// TIA Portal V16 export
// export: Created 2023-05-15T10:42:05.211121Z, ExportSetting WithDefaults, DisplayName Totally Integrated Automation Portal, DisplayVersion V16 Update 3, DisplayName TIA Portal Version Control Interface, DisplayVersion V16 Update 2, DisplayName TIA Portal Openness, DisplayVersion V16 Update 3, DisplayName SINAMICS Startdrive Advanced, DisplayVersion V16, DisplayName SINAMICS Startdrive G130, G150, S120, S150, SINAMICS MV, S210, DisplayVersion V16, DisplayName SINAMICS Startdrive G110M, G120, G120C, G120D, G120P, DisplayVersion V16, DisplayName STEP 7 Professional, DisplayVersion V16 Update 3, DisplayName STEP 7 Safety, DisplayVersion V16, DisplayName WinCC Advanced, DisplayVersion V16 Update 3
FUNCTION "AUTO_HBA2" : Void   // FC45, LAD
{ S7_Optimized_Access := 'FALSE' }
VERSION : 0.1
// prueba con paco de comit 2 b
// 1040 desde paco
// stored: AutoNumber false, IsIECCheckEnabled false, SetENOAutomatically false, UDAEnableTagReadback false
   VAR_TEMP
      SEGUIR : Bool;
      aux_int_1 : Int;
      TEMP0 : Bool;
   END_VAR
   VAR_TEMP   // added for the SCL form of the ladder/FBD networks
      _w1 : Bool;
      _s5time1 : S5Time;
   END_VAR
BEGIN

REGION Network 1: ACTIVACION VAN300
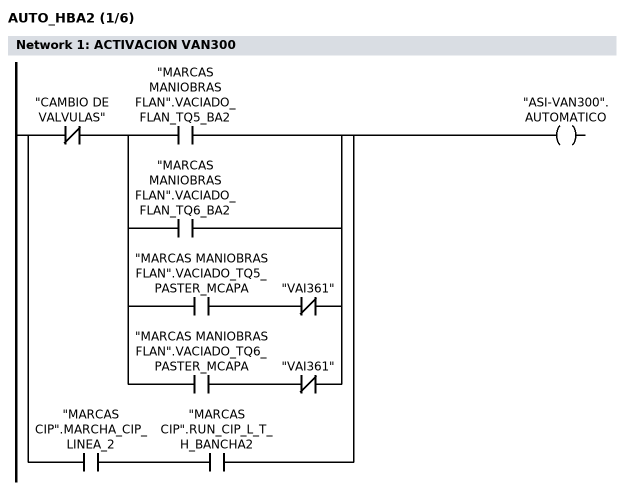
   RUNG wire#powerrail
      I_Contact( "CAMBIO DE VALVULAS" )
      wire#w1
      Contact( "MARCAS MANIOBRAS FLAN".VACIADO_FLAN_TQ5_BA2 )
      wire#w2
      Coil( "ASI-VAN300".AUTOMATICO )
   END_RUNG
   RUNG wire#w1
      Contact( "MARCAS MANIOBRAS FLAN".VACIADO_FLAN_TQ6_BA2 )
   END_RUNG wire#w2
   RUNG wire#w1
      Contact( "MARCAS MANIOBRAS FLAN".VACIADO_TQ5_PASTER_MCAPA )
      I_Contact( "VAI361" )
   END_RUNG wire#w2
   RUNG wire#w1
      Contact( "MARCAS MANIOBRAS FLAN".VACIADO_TQ6_PASTER_MCAPA )
      I_Contact( "VAI361" )
   END_RUNG wire#w2
   RUNG wire#powerrail
      Contact( "MARCAS CIP".MARCHA_CIP_LINEA_2 )
      Contact( "MARCAS CIP".RUN_CIP_L_T_H_BANCHA2 )
   END_RUNG wire#w2
   // the same network as SCL:
   "ASI-VAN300".AUTOMATICO := (NOT "CAMBIO DE VALVULAS" AND ("MARCAS MANIOBRAS FLAN".VACIADO_FLAN_TQ5_BA2 OR "MARCAS MANIOBRAS FLAN".VACIADO_FLAN_TQ6_BA2 OR ("MARCAS MANIOBRAS FLAN".VACIADO_TQ5_PASTER_MCAPA AND NOT "VAI361") OR ("MARCAS MANIOBRAS FLAN".VACIADO_TQ6_PASTER_MCAPA AND NOT "VAI361"))) OR ("MARCAS CIP".MARCHA_CIP_LINEA_2 AND "MARCAS CIP".RUN_CIP_L_T_H_BANCHA2);
END_REGION

REGION Network 2: ACTIVACION VMN301
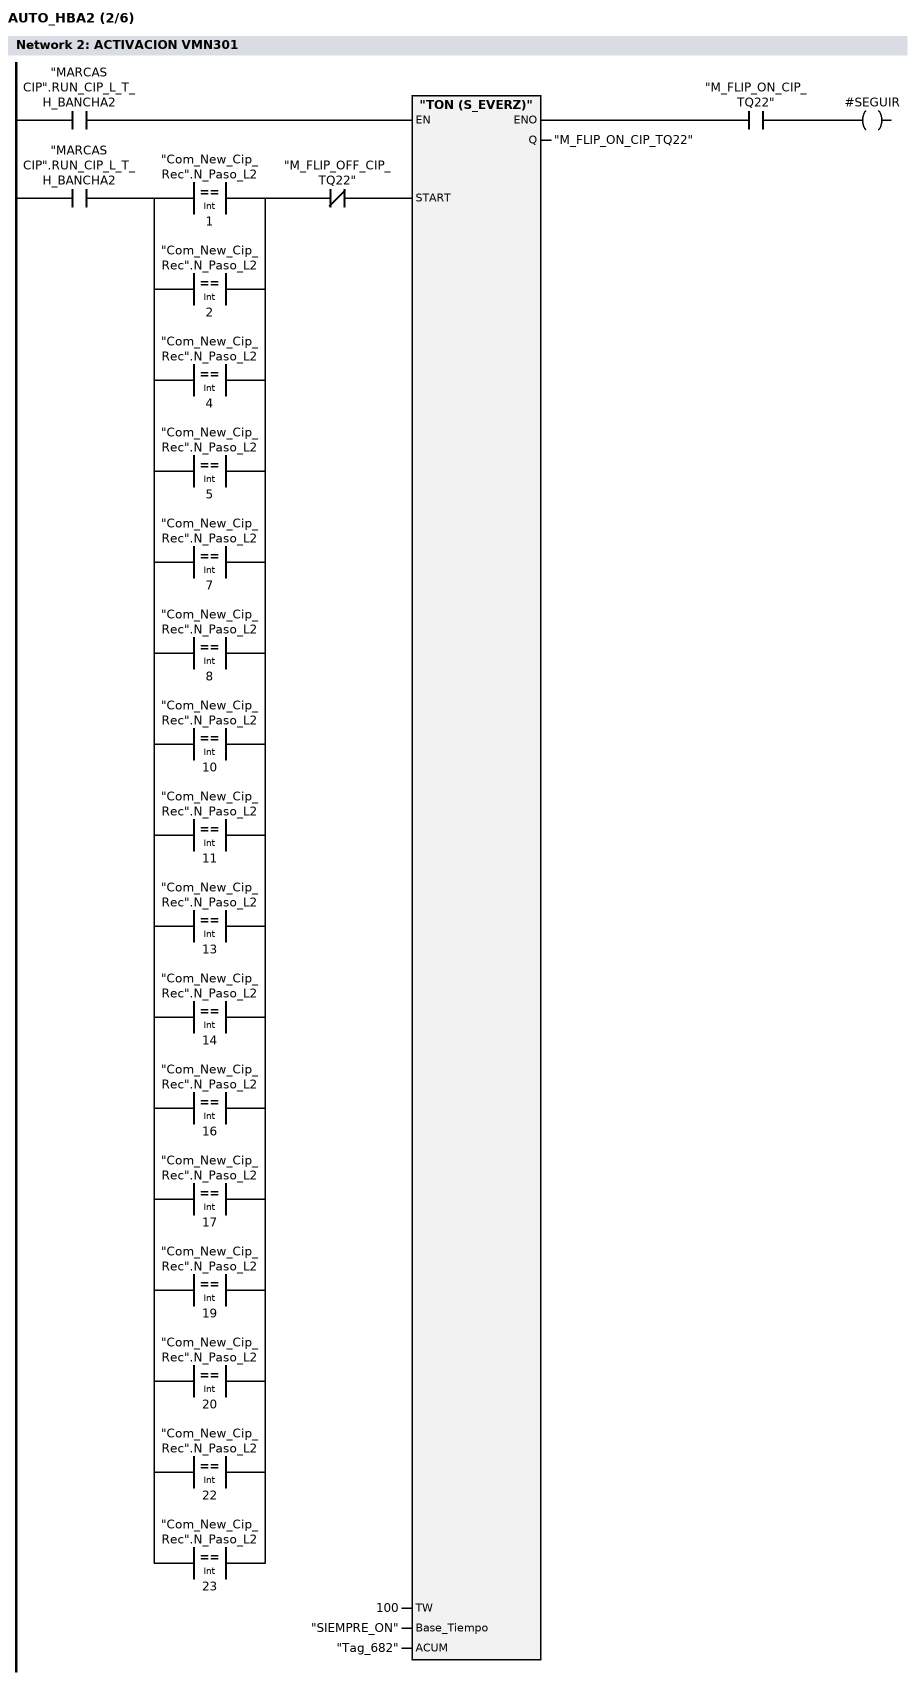
   RUNG wire#powerrail
      Contact( "MARCAS CIP".RUN_CIP_L_T_H_BANCHA2 )
      "TON (S_EVERZ)"(TW := 100, Base_Tiempo := "SIEMPRE_ON", Q => "M_FLIP_ON_CIP_TQ22", ACUM := "Tag_682", START := wire#w3)
      Contact( "M_FLIP_ON_CIP_TQ22" )
      Coil( #SEGUIR )
   END_RUNG
   RUNG wire#powerrail
      Contact( "MARCAS CIP".RUN_CIP_L_T_H_BANCHA2 )
      wire#w1
      { S7_Templates := "SrcType := Int" } EQ_Contact(in1 := "Com_New_Cip_Rec".N_Paso_L2, in2 := 1)
      wire#w2
      I_Contact( "M_FLIP_OFF_CIP_TQ22" )
   END_RUNG wire#w3
   RUNG wire#w1
      { S7_Templates := "SrcType := Int" } EQ_Contact(in1 := "Com_New_Cip_Rec".N_Paso_L2, in2 := 2)
   END_RUNG wire#w2
   RUNG wire#w1
      { S7_Templates := "SrcType := Int" } EQ_Contact(in1 := "Com_New_Cip_Rec".N_Paso_L2, in2 := 4)
   END_RUNG wire#w2
   RUNG wire#w1
      { S7_Templates := "SrcType := Int" } EQ_Contact(in1 := "Com_New_Cip_Rec".N_Paso_L2, in2 := 5)
   END_RUNG wire#w2
   RUNG wire#w1
      { S7_Templates := "SrcType := Int" } EQ_Contact(in1 := "Com_New_Cip_Rec".N_Paso_L2, in2 := 7)
   END_RUNG wire#w2
   RUNG wire#w1
      { S7_Templates := "SrcType := Int" } EQ_Contact(in1 := "Com_New_Cip_Rec".N_Paso_L2, in2 := 8)
   END_RUNG wire#w2
   RUNG wire#w1
      { S7_Templates := "SrcType := Int" } EQ_Contact(in1 := "Com_New_Cip_Rec".N_Paso_L2, in2 := 10)
   END_RUNG wire#w2
   RUNG wire#w1
      { S7_Templates := "SrcType := Int" } EQ_Contact(in1 := "Com_New_Cip_Rec".N_Paso_L2, in2 := 11)
   END_RUNG wire#w2
   RUNG wire#w1
      { S7_Templates := "SrcType := Int" } EQ_Contact(in1 := "Com_New_Cip_Rec".N_Paso_L2, in2 := 13)
   END_RUNG wire#w2
   RUNG wire#w1
      { S7_Templates := "SrcType := Int" } EQ_Contact(in1 := "Com_New_Cip_Rec".N_Paso_L2, in2 := 14)
   END_RUNG wire#w2
   RUNG wire#w1
      { S7_Templates := "SrcType := Int" } EQ_Contact(in1 := "Com_New_Cip_Rec".N_Paso_L2, in2 := 16)
   END_RUNG wire#w2
   RUNG wire#w1
      { S7_Templates := "SrcType := Int" } EQ_Contact(in1 := "Com_New_Cip_Rec".N_Paso_L2, in2 := 17)
   END_RUNG wire#w2
   RUNG wire#w1
      { S7_Templates := "SrcType := Int" } EQ_Contact(in1 := "Com_New_Cip_Rec".N_Paso_L2, in2 := 19)
   END_RUNG wire#w2
   RUNG wire#w1
      { S7_Templates := "SrcType := Int" } EQ_Contact(in1 := "Com_New_Cip_Rec".N_Paso_L2, in2 := 20)
   END_RUNG wire#w2
   RUNG wire#w1
      { S7_Templates := "SrcType := Int" } EQ_Contact(in1 := "Com_New_Cip_Rec".N_Paso_L2, in2 := 22)
   END_RUNG wire#w2
   RUNG wire#w1
      { S7_Templates := "SrcType := Int" } EQ_Contact(in1 := "Com_New_Cip_Rec".N_Paso_L2, in2 := 23)
   END_RUNG wire#w2
   // the same network as SCL:
   "TON (S_EVERZ)"(EN := "MARCAS CIP".RUN_CIP_L_T_H_BANCHA2,
                   START := "MARCAS CIP".RUN_CIP_L_T_H_BANCHA2 AND (("Com_New_Cip_Rec".N_Paso_L2 = 1) OR ("Com_New_Cip_Rec".N_Paso_L2 = 2) OR ("Com_New_Cip_Rec".N_Paso_L2 = 4) OR ("Com_New_Cip_Rec".N_Paso_L2 = 5) OR ("Com_New_Cip_Rec".N_Paso_L2 = 7) OR ("Com_New_Cip_Rec".N_Paso_L2 = 8) OR ("Com_New_Cip_Rec".N_Paso_L2 = 10) OR ("Com_New_Cip_Rec".N_Paso_L2 = 11) OR ("Com_New_Cip_Rec".N_Paso_L2 = 13) OR ("Com_New_Cip_Rec".N_Paso_L2 = 14) OR ("Com_New_Cip_Rec".N_Paso_L2 = 16) OR ("Com_New_Cip_Rec".N_Paso_L2 = 17) OR ("Com_New_Cip_Rec".N_Paso_L2 = 19) OR ("Com_New_Cip_Rec".N_Paso_L2 = 20) OR ("Com_New_Cip_Rec".N_Paso_L2 = 22) OR ("Com_New_Cip_Rec".N_Paso_L2 = 23)) AND NOT "M_FLIP_OFF_CIP_TQ22",
                   TW := 100,
                   Base_Tiempo := "SIEMPRE_ON",
                   ACUM := "Tag_682",
                   Q => "M_FLIP_ON_CIP_TQ22",
                   ENO => #_w1);
   #SEGUIR := #_w1 AND "M_FLIP_ON_CIP_TQ22";
END_REGION

REGION Network 3
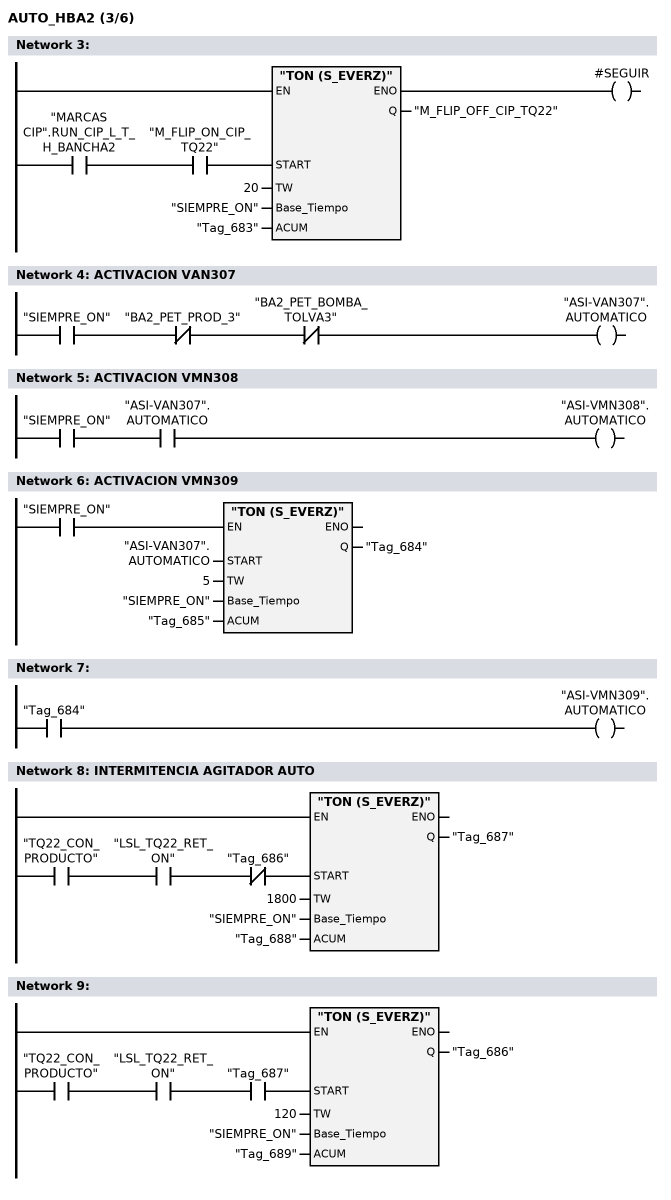
   RUNG wire#powerrail
      "TON (S_EVERZ)"(TW := 20, Base_Tiempo := "SIEMPRE_ON", Q => "M_FLIP_OFF_CIP_TQ22", ACUM := "Tag_683", START := wire#w1)
      Coil( #SEGUIR )
   END_RUNG
   RUNG wire#powerrail
      Contact( "MARCAS CIP".RUN_CIP_L_T_H_BANCHA2 )
      Contact( "M_FLIP_ON_CIP_TQ22" )
   END_RUNG wire#w1
   // the same network as SCL:
   "TON (S_EVERZ)"(START := "MARCAS CIP".RUN_CIP_L_T_H_BANCHA2 AND "M_FLIP_ON_CIP_TQ22",
                   TW := 20,
                   Base_Tiempo := "SIEMPRE_ON",
                   ACUM := "Tag_683",
                   Q => "M_FLIP_OFF_CIP_TQ22",
                   ENO => #_w1);
   #SEGUIR := #_w1;
END_REGION

REGION Network 4: ACTIVACION VAN307
   RUNG wire#powerrail
      Contact( "SIEMPRE_ON" )
      I_Contact( "BA2_PET_PROD_3" )
      I_Contact( "BA2_PET_BOMBA_TOLVA3" )
      Coil( "ASI-VAN307".AUTOMATICO )
   END_RUNG
   // the same network as SCL:
   "ASI-VAN307".AUTOMATICO := "SIEMPRE_ON" AND NOT "BA2_PET_PROD_3" AND NOT "BA2_PET_BOMBA_TOLVA3";
END_REGION

REGION Network 5: ACTIVACION VMN308
   RUNG wire#powerrail
      Contact( "SIEMPRE_ON" )
      Contact( "ASI-VAN307".AUTOMATICO )
      Coil( "ASI-VMN308".AUTOMATICO )
   END_RUNG
   // the same network as SCL:
   "ASI-VMN308".AUTOMATICO := "SIEMPRE_ON" AND "ASI-VAN307".AUTOMATICO;
END_REGION

REGION Network 6: ACTIVACION VMN309
   RUNG wire#powerrail
      Contact( "SIEMPRE_ON" )
      "TON (S_EVERZ)"(START := "ASI-VAN307".AUTOMATICO, TW := 5, Base_Tiempo := "SIEMPRE_ON", Q => "Tag_684", ACUM := "Tag_685")
   END_RUNG
   // the same network as SCL:
   IF "SIEMPRE_ON" THEN
       "TON (S_EVERZ)"(START := "ASI-VAN307".AUTOMATICO,
                       TW := 5,
                       Base_Tiempo := "SIEMPRE_ON",
                       ACUM := "Tag_685",
                       Q => "Tag_684");
   END_IF;
END_REGION

REGION Network 7
   RUNG wire#powerrail
      Contact( "Tag_684" )
      Coil( "ASI-VMN309".AUTOMATICO )
   END_RUNG
   // the same network as SCL:
   "ASI-VMN309".AUTOMATICO := "Tag_684";
END_REGION

REGION Network 8: INTERMITENCIA AGITADOR AUTO
   RUNG wire#powerrail
      "TON (S_EVERZ)"(TW := 1800, Base_Tiempo := "SIEMPRE_ON", Q => "Tag_687", ACUM := "Tag_688", START := wire#w1)
   END_RUNG
   RUNG wire#powerrail
      Contact( "TQ22_CON_PRODUCTO" )
      Contact( "LSL_TQ22_RET_ON" )
      I_Contact( "Tag_686" )
   END_RUNG wire#w1
   // the same network as SCL:
   "TON (S_EVERZ)"(START := "TQ22_CON_PRODUCTO" AND "LSL_TQ22_RET_ON" AND NOT "Tag_686",
                   TW := 1800,
                   Base_Tiempo := "SIEMPRE_ON",
                   ACUM := "Tag_688",
                   Q => "Tag_687");
END_REGION

REGION Network 9
   RUNG wire#powerrail
      "TON (S_EVERZ)"(TW := 120, Base_Tiempo := "SIEMPRE_ON", Q => "Tag_686", ACUM := "Tag_689", START := wire#w1)
   END_RUNG
   RUNG wire#powerrail
      Contact( "TQ22_CON_PRODUCTO" )
      Contact( "LSL_TQ22_RET_ON" )
      Contact( "Tag_687" )
   END_RUNG wire#w1
   // the same network as SCL:
   "TON (S_EVERZ)"(START := "TQ22_CON_PRODUCTO" AND "LSL_TQ22_RET_ON" AND "Tag_687",
                   TW := 120,
                   Base_Tiempo := "SIEMPRE_ON",
                   ACUM := "Tag_689",
                   Q => "Tag_686");
END_REGION

REGION Network 10: ACTIVACION AGITADOR TQ22 (NUEVO)
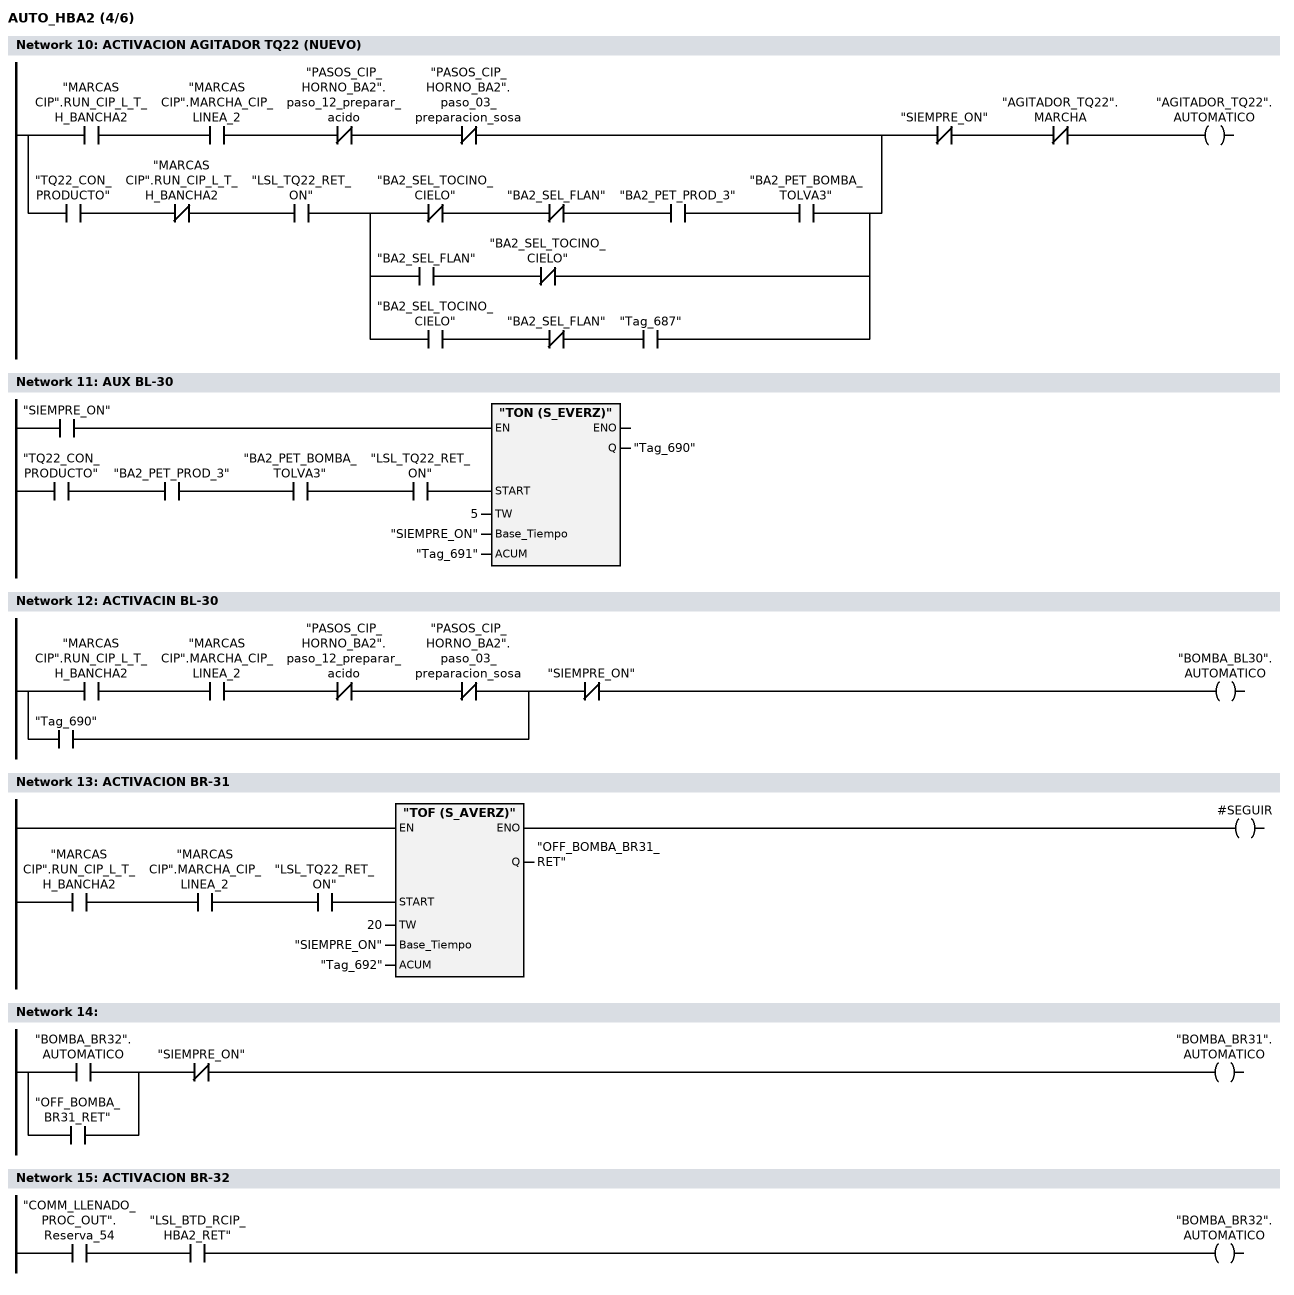
   RUNG wire#powerrail
      Contact( "MARCAS CIP".RUN_CIP_L_T_H_BANCHA2 )
      Contact( "MARCAS CIP".MARCHA_CIP_LINEA_2 )
      I_Contact( "PASOS_CIP_HORNO_BA2".paso_12_preparar_acido )
      I_Contact( "PASOS_CIP_HORNO_BA2".paso_03_preparacion_sosa )
      wire#w1
      I_Contact( "SIEMPRE_ON" )
      I_Contact( "AGITADOR_TQ22".MARCHA )
      Coil( "AGITADOR_TQ22".AUTOMATICO )
   END_RUNG
   RUNG wire#powerrail
      Contact( "TQ22_CON_PRODUCTO" )
      I_Contact( "MARCAS CIP".RUN_CIP_L_T_H_BANCHA2 )
      Contact( "LSL_TQ22_RET_ON" )
      wire#w2
      I_Contact( "BA2_SEL_TOCINO_CIELO" )
      I_Contact( "BA2_SEL_FLAN" )
      Contact( "BA2_PET_PROD_3" )
      Contact( "BA2_PET_BOMBA_TOLVA3" )
   END_RUNG wire#w1
   RUNG wire#w2
      Contact( "BA2_SEL_FLAN" )
      I_Contact( "BA2_SEL_TOCINO_CIELO" )
   END_RUNG wire#w1
   RUNG wire#w2
      Contact( "BA2_SEL_TOCINO_CIELO" )
      I_Contact( "BA2_SEL_FLAN" )
      Contact( "Tag_687" )
   END_RUNG wire#w1
   // the same network as SCL:
   "AGITADOR_TQ22".AUTOMATICO := (("MARCAS CIP".RUN_CIP_L_T_H_BANCHA2 AND "MARCAS CIP".MARCHA_CIP_LINEA_2 AND NOT "PASOS_CIP_HORNO_BA2".paso_12_preparar_acido AND NOT "PASOS_CIP_HORNO_BA2".paso_03_preparacion_sosa) OR ("TQ22_CON_PRODUCTO" AND NOT "MARCAS CIP".RUN_CIP_L_T_H_BANCHA2 AND "LSL_TQ22_RET_ON" AND ((NOT "BA2_SEL_TOCINO_CIELO" AND NOT "BA2_SEL_FLAN" AND "BA2_PET_PROD_3" AND "BA2_PET_BOMBA_TOLVA3") OR ("BA2_SEL_FLAN" AND NOT "BA2_SEL_TOCINO_CIELO") OR ("BA2_SEL_TOCINO_CIELO" AND NOT "BA2_SEL_FLAN" AND "Tag_687")))) AND NOT "SIEMPRE_ON" AND NOT "AGITADOR_TQ22".MARCHA;
END_REGION

REGION Network 11: AUX BL-30
   RUNG wire#powerrail
      Contact( "SIEMPRE_ON" )
      "TON (S_EVERZ)"(TW := 5, Base_Tiempo := "SIEMPRE_ON", Q => "Tag_690", ACUM := "Tag_691", START := wire#w1)
   END_RUNG
   RUNG wire#powerrail
      Contact( "TQ22_CON_PRODUCTO" )
      Contact( "BA2_PET_PROD_3" )
      Contact( "BA2_PET_BOMBA_TOLVA3" )
      Contact( "LSL_TQ22_RET_ON" )
   END_RUNG wire#w1
   // the same network as SCL:
   IF "SIEMPRE_ON" THEN
       "TON (S_EVERZ)"(START := "TQ22_CON_PRODUCTO" AND "BA2_PET_PROD_3" AND "BA2_PET_BOMBA_TOLVA3" AND "LSL_TQ22_RET_ON",
                       TW := 5,
                       Base_Tiempo := "SIEMPRE_ON",
                       ACUM := "Tag_691",
                       Q => "Tag_690");
   END_IF;
END_REGION

REGION Network 12: ACTIVACIN BL-30
   RUNG wire#powerrail
      Contact( "MARCAS CIP".RUN_CIP_L_T_H_BANCHA2 )
      Contact( "MARCAS CIP".MARCHA_CIP_LINEA_2 )
      I_Contact( "PASOS_CIP_HORNO_BA2".paso_12_preparar_acido )
      I_Contact( "PASOS_CIP_HORNO_BA2".paso_03_preparacion_sosa )
      wire#w1
      I_Contact( "SIEMPRE_ON" )
      Coil( "BOMBA_BL30".AUTOMATICO )
   END_RUNG
   RUNG wire#powerrail
      Contact( "Tag_690" )
   END_RUNG wire#w1
   // the same network as SCL:
   "BOMBA_BL30".AUTOMATICO := (("MARCAS CIP".RUN_CIP_L_T_H_BANCHA2 AND "MARCAS CIP".MARCHA_CIP_LINEA_2 AND NOT "PASOS_CIP_HORNO_BA2".paso_12_preparar_acido AND NOT "PASOS_CIP_HORNO_BA2".paso_03_preparacion_sosa) OR "Tag_690") AND NOT "SIEMPRE_ON";
END_REGION

REGION Network 13: ACTIVACION BR-31
   RUNG wire#powerrail
      "TOF (S_AVERZ)"(TW := 20, Base_Tiempo := "SIEMPRE_ON", Q => "OFF_BOMBA_BR31_RET", ACUM := "Tag_692", START := wire#w1)
      Coil( #SEGUIR )
   END_RUNG
   RUNG wire#powerrail
      Contact( "MARCAS CIP".RUN_CIP_L_T_H_BANCHA2 )
      Contact( "MARCAS CIP".MARCHA_CIP_LINEA_2 )
      Contact( "LSL_TQ22_RET_ON" )
   END_RUNG wire#w1
   // the same network as SCL:
   "TOF (S_AVERZ)"(START := "MARCAS CIP".RUN_CIP_L_T_H_BANCHA2 AND "MARCAS CIP".MARCHA_CIP_LINEA_2 AND "LSL_TQ22_RET_ON",
                   TW := 20,
                   Base_Tiempo := "SIEMPRE_ON",
                   ACUM := "Tag_692",
                   Q => "OFF_BOMBA_BR31_RET",
                   ENO => #_w1);
   #SEGUIR := #_w1;
END_REGION

REGION Network 14
   RUNG wire#powerrail
      Contact( "BOMBA_BR32".AUTOMATICO )
      wire#w1
      I_Contact( "SIEMPRE_ON" )
      Coil( "BOMBA_BR31".AUTOMATICO )
   END_RUNG
   RUNG wire#powerrail
      Contact( "OFF_BOMBA_BR31_RET" )
   END_RUNG wire#w1
   // the same network as SCL:
   "BOMBA_BR31".AUTOMATICO := ("BOMBA_BR32".AUTOMATICO OR "OFF_BOMBA_BR31_RET") AND NOT "SIEMPRE_ON";
END_REGION

REGION Network 15: ACTIVACION BR-32
   RUNG wire#powerrail
      Contact( "COMM_LLENADO_PROC_OUT".Reserva_54 )
      Contact( "LSL_BTD_RCIP_HBA2_RET" )
      Coil( "BOMBA_BR32".AUTOMATICO )
   END_RUNG
   // the same network as SCL:
   "BOMBA_BR32".AUTOMATICO := "COMM_LLENADO_PROC_OUT".Reserva_54 AND "LSL_BTD_RCIP_HBA2_RET";
END_REGION

REGION Network 16: ACTIVACION BL-33 BOMBA DE CARAMELO
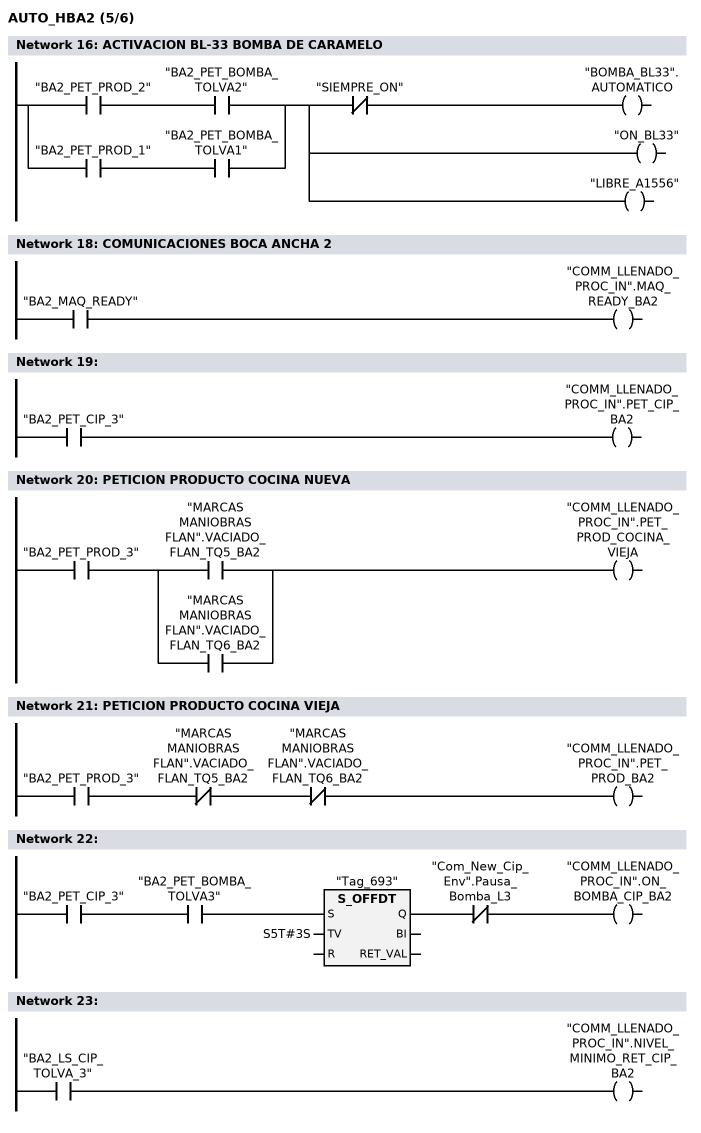
   RUNG wire#powerrail
      Contact( "BA2_PET_PROD_2" )
      Contact( "BA2_PET_BOMBA_TOLVA2" )
      wire#w1
      I_Contact( "SIEMPRE_ON" )
      Coil( "BOMBA_BL33".AUTOMATICO )
   END_RUNG
   RUNG wire#powerrail
      Contact( "BA2_PET_PROD_1" )
      Contact( "BA2_PET_BOMBA_TOLVA1" )
   END_RUNG wire#w1
   RUNG wire#w1
      Coil( "ON_BL33" )
   END_RUNG
   RUNG wire#w1
      Coil( "LIBRE_A1556" )
   END_RUNG
   // the same network as SCL:
   #_w1 := ("BA2_PET_PROD_2" AND "BA2_PET_BOMBA_TOLVA2") OR ("BA2_PET_PROD_1" AND "BA2_PET_BOMBA_TOLVA1");
   "BOMBA_BL33".AUTOMATICO := #_w1 AND NOT "SIEMPRE_ON";
   "ON_BL33" := #_w1;
   "LIBRE_A1556" := #_w1;
END_REGION

REGION Network 17: VACIO
END_REGION

REGION Network 18: COMUNICACIONES BOCA ANCHA 2
   RUNG wire#powerrail
      Contact( "BA2_MAQ_READY" )
      Coil( "COMM_LLENADO_PROC_IN".MAQ_READY_BA2 )
   END_RUNG
   // the same network as SCL:
   "COMM_LLENADO_PROC_IN".MAQ_READY_BA2 := "BA2_MAQ_READY";
END_REGION

REGION Network 19
   RUNG wire#powerrail
      Contact( "BA2_PET_CIP_3" )
      Coil( "COMM_LLENADO_PROC_IN".PET_CIP_BA2 )
   END_RUNG
   // the same network as SCL:
   "COMM_LLENADO_PROC_IN".PET_CIP_BA2 := "BA2_PET_CIP_3";
END_REGION

REGION Network 20: PETICION PRODUCTO COCINA NUEVA
   RUNG wire#powerrail
      Contact( "BA2_PET_PROD_3" )
      wire#w1
      Contact( "MARCAS MANIOBRAS FLAN".VACIADO_FLAN_TQ5_BA2 )
      wire#w2
      Coil( "COMM_LLENADO_PROC_IN".PET_PROD_COCINA_VIEJA )
   END_RUNG
   RUNG wire#w1
      Contact( "MARCAS MANIOBRAS FLAN".VACIADO_FLAN_TQ6_BA2 )
   END_RUNG wire#w2
   // the same network as SCL:
   "COMM_LLENADO_PROC_IN".PET_PROD_COCINA_VIEJA := "BA2_PET_PROD_3" AND ("MARCAS MANIOBRAS FLAN".VACIADO_FLAN_TQ5_BA2 OR "MARCAS MANIOBRAS FLAN".VACIADO_FLAN_TQ6_BA2);
END_REGION

REGION Network 21: PETICION PRODUCTO COCINA VIEJA
   RUNG wire#powerrail
      Contact( "BA2_PET_PROD_3" )
      I_Contact( "MARCAS MANIOBRAS FLAN".VACIADO_FLAN_TQ5_BA2 )
      I_Contact( "MARCAS MANIOBRAS FLAN".VACIADO_FLAN_TQ6_BA2 )
      Coil( "COMM_LLENADO_PROC_IN".PET_PROD_BA2 )
   END_RUNG
   // the same network as SCL:
   "COMM_LLENADO_PROC_IN".PET_PROD_BA2 := "BA2_PET_PROD_3" AND NOT "MARCAS MANIOBRAS FLAN".VACIADO_FLAN_TQ5_BA2 AND NOT "MARCAS MANIOBRAS FLAN".VACIADO_FLAN_TQ6_BA2;
END_REGION

REGION Network 22
   RUNG wire#powerrail
      Contact( "BA2_PET_CIP_3" )
      Contact( "BA2_PET_BOMBA_TOLVA3" )
      S_OFFDT(T_NO := "Tag_693", TV := S5T#3S, R :=, BI =>, RET_VAL =>)
      I_Contact( "Com_New_Cip_Env".Pausa_Bomba_L3 )
      Coil( "COMM_LLENADO_PROC_IN".ON_BOMBA_CIP_BA2 )
   END_RUNG
   // the same network as SCL:
   #_s5time1 := S_OFFDT(T_NO := "Tag_693",
                        TV := S5T#3S,
                        S := "BA2_PET_CIP_3" AND "BA2_PET_BOMBA_TOLVA3",
                        Q => #_w1);
   "COMM_LLENADO_PROC_IN".ON_BOMBA_CIP_BA2 := #_w1 AND NOT "Com_New_Cip_Env".Pausa_Bomba_L3;
END_REGION

REGION Network 23
   RUNG wire#powerrail
      Contact( "BA2_LS_CIP_TOLVA_3" )
      Coil( "COMM_LLENADO_PROC_IN".NIVEL_MINIMO_RET_CIP_BA2 )
   END_RUNG
   // the same network as SCL:
   "COMM_LLENADO_PROC_IN".NIVEL_MINIMO_RET_CIP_BA2 := "BA2_LS_CIP_TOLVA_3";
END_REGION

REGION Network 24: BIT PERMISO ENVIO BA2
   // SE ANULA LINEA POR QUE LA LIMPIEZA PARA EL ENVIO DE PRODUCTO A BA2
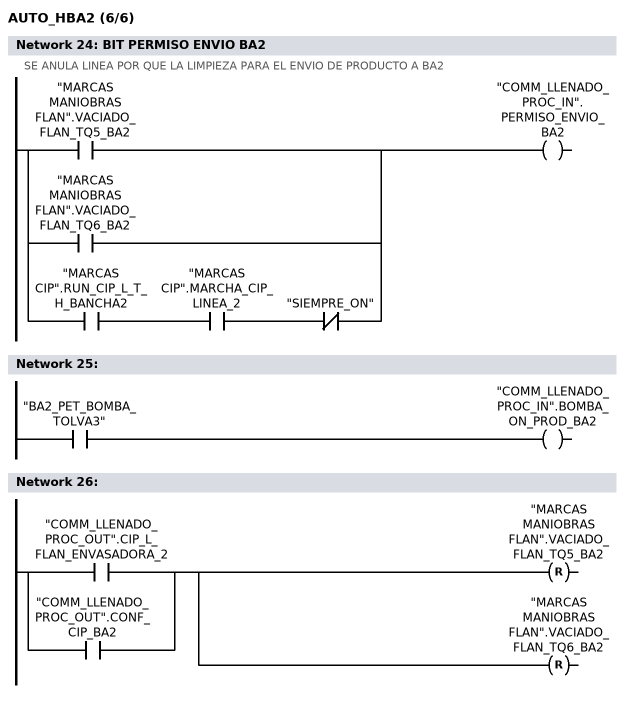
   RUNG wire#powerrail
      Contact( "MARCAS MANIOBRAS FLAN".VACIADO_FLAN_TQ5_BA2 )
      wire#w1
      Coil( "COMM_LLENADO_PROC_IN".PERMISO_ENVIO_BA2 )
   END_RUNG
   RUNG wire#powerrail
      Contact( "MARCAS MANIOBRAS FLAN".VACIADO_FLAN_TQ6_BA2 )
   END_RUNG wire#w1
   RUNG wire#powerrail
      Contact( "MARCAS CIP".RUN_CIP_L_T_H_BANCHA2 )
      Contact( "MARCAS CIP".MARCHA_CIP_LINEA_2 )
      I_Contact( "SIEMPRE_ON" )
   END_RUNG wire#w1
   // the same network as SCL:
   "COMM_LLENADO_PROC_IN".PERMISO_ENVIO_BA2 := "MARCAS MANIOBRAS FLAN".VACIADO_FLAN_TQ5_BA2 OR "MARCAS MANIOBRAS FLAN".VACIADO_FLAN_TQ6_BA2 OR ("MARCAS CIP".RUN_CIP_L_T_H_BANCHA2 AND "MARCAS CIP".MARCHA_CIP_LINEA_2 AND NOT "SIEMPRE_ON");
END_REGION

REGION Network 25
   RUNG wire#powerrail
      Contact( "BA2_PET_BOMBA_TOLVA3" )
      Coil( "COMM_LLENADO_PROC_IN".BOMBA_ON_PROD_BA2 )
   END_RUNG
   // the same network as SCL:
   "COMM_LLENADO_PROC_IN".BOMBA_ON_PROD_BA2 := "BA2_PET_BOMBA_TOLVA3";
END_REGION

REGION Network 26
   RUNG wire#powerrail
      Contact( "COMM_LLENADO_PROC_OUT".CIP_L_FLAN_ENVASADORA_2 )
      wire#w1
      R_Coil( "MARCAS MANIOBRAS FLAN".VACIADO_FLAN_TQ5_BA2 )
   END_RUNG
   RUNG wire#powerrail
      Contact( "COMM_LLENADO_PROC_OUT".CONF_CIP_BA2 )
   END_RUNG wire#w1
   RUNG wire#w1
      R_Coil( "MARCAS MANIOBRAS FLAN".VACIADO_FLAN_TQ6_BA2 )
   END_RUNG
   // the same network as SCL:
   IF "COMM_LLENADO_PROC_OUT".CIP_L_FLAN_ENVASADORA_2 OR "COMM_LLENADO_PROC_OUT".CONF_CIP_BA2 THEN
       "MARCAS MANIOBRAS FLAN".VACIADO_FLAN_TQ5_BA2 := FALSE;
       "MARCAS MANIOBRAS FLAN".VACIADO_FLAN_TQ6_BA2 := FALSE;
   END_IF;
END_REGION
END_FUNCTION
